// Mitsubishi GX Works2 project: a12   PLC: Q02/Q02H

PROGRAM MAIN
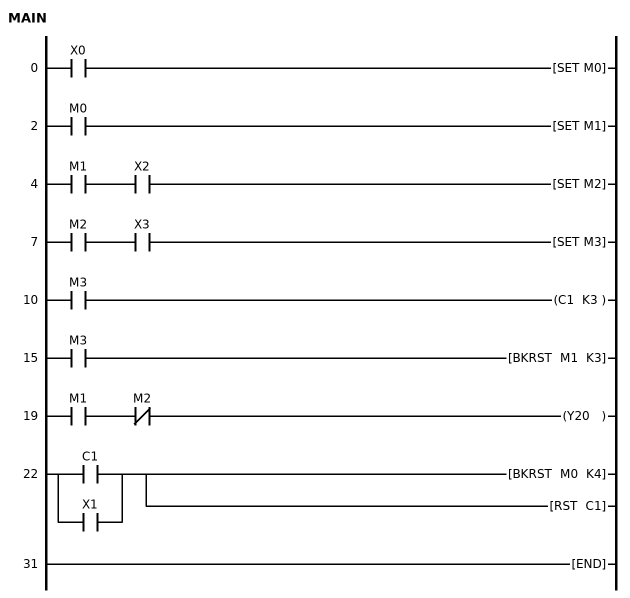
0     LD      X0
      SET     M0
2     LD      M0
      SET     M1
4     LD      M1
      AND     X2
      SET     M2
7     LD      M2
      AND     X3
      SET     M3
10    LD      M3
      OUT     C1 K3
15    LD      M3
      BKRST   M1 K3
19    LD      M1
      ANI     M2
      OUT     Y20
22    LD      C1
      OR      X1
      BKRST   M0 K4
      RST     C1
31    END
END_PROGRAM
